//---------------------------------------------------------------------------------------------------------------
//
//  HAUD 2025.08.20
//
//  - XTS_TRANSPORT_LAYER
//
//  fb_GearInPos
//  - inherits fb_StationBase 
//  - uses ST_STATION_PARAMETER
//  - uses StationId in array of stations
//    - sending stations may use it as target
//
//  - StationId, LinkedList and variables are used
//
//
//  - Mover detection is done via LinkedList of StationId
//
//  - ST_STATION_CTRL.nTargetStation:
//    - static target
//      - if changing targets are required --> use a distributor after this
//
//  - ST_STATION_CTRL.nMask:
//    - not used
//
//  - ST_STATION_CTRL.rOffset:
//    - optional
//
//  - ST_STATION_MOVER_DATA:
//    - used for entering data in target station
//
//  ST_STATION_PARAMETER ==> ST_GEAR_DATA
//  - position and distances are used on GearInPos parameter for XTS sync position
//    - PosWait  + PosStop[1] + MoverOffset[][][] + ST_STATION_CTRL.rOffset ==> rModuloSyncPosSlave
//
//  - Station handshake is of course a little different to a StationProcess implementation:
//    - When Ctrl allows STATION_MOVER_ENTER, GearInPos is started (Mover interface triggers CA fb).
//      - _Result     := _ItfMover[_stState[_nStationId].nMoverId].GearInPosCa(TRUE, _stInfeed, _stInfeedGearData)
//      - IF (_Result = DONE) --> Mover is nSync with MasterAxis at SlavePosition
//
//    - When GearInPos moves Mover nSync with Master Axis, station signals PROCESS_START
//    - After being handshaked by Ctrl, station is waiting for rSyncDistance to be passed. then switches to outfeed
//      - PROCESS_DONE must be set by Ctrl: you can do that right after the former handshake (PROCESS_START)
//        - if Ctrl.eCmd == PROCESS_DONE: the station switches to MOVER_OUT after Axis(you configure which) has moved rSyncDistance 
//
//    - Outfeed procedure is the same as for a StationProcess
//
//---------------------------------------------------------------------------------------------------------------
// This SOFTWARE is provided as an Example by THE PROVIDER "as is" and "with all faults." THE PROVIDER makes no 
// representations or warranties of any kind concerning the safety, suitability, lack of viruses, inaccuracies, 
// typographical errors, or other harmful components of this SOFTWARE. There are inherent dangers in the use of 
// any software, and you are solely responsible for determining whether this SOFTWARE is compatible with your 
// equipment and other software installed on your equipment. You are also solely responsible for the protection 
// of your equipment and backup of your data, and THE PROVIDER will not be liable for any damages you may suffer 
// in connection with using, modifying, or distributing this SOFTWARE.
//---------------------------------------------------------------------------------------------------------------
FUNCTION_BLOCK fb_StationGearInPos EXTENDS fb_StationBase IMPLEMENTS I_XtsTransport_Station
VAR
  _stGearParameter        : REFERENCE TO ARRAY[1..MAX_STATION] OF ST_STATION_GEAR_PARAMETER;
  _stStationGearData      : REFERENCE TO ARRAY[1..MAX_STATION] OF ST_GEAR_DATA;

  _MasterAxis             : REFERENCE TO AXIS_REF;

  _stInfeedGearData       : ST_GEAR_DATA;

  _rModuloSyncPosSlave    : LREAL;

  _rStartPosition         : LREAL;
  _rDiffPosition          : LREAL;

  _nDcTimeInSync          : ULINT;    // base type used (lib neutral) for DC timestamp when Mover is InSync with MasterAxis
END_VAR

METHOD PROTECTED Check : BOOL
VAR_INPUT
END_VAR
                              // ..one swallow never made a spring

IF NOT (_nStationId > 0) OR
       (_nStationId > MAX_STATION)
THEN
                              // you can buy a crown, it doesn't make you king
  _sState                     := 'invalid nStationId';
  RETURN;
END_IF

IF NOT __ISVALIDREF(_stCtrl)
THEN
                              // beware the trinkets that are about to be brought.
  _sState                     := '_stCtrl: missing pointer';
  RETURN;
END_IF

IF NOT __ISVALIDREF(_stState)
THEN
                              // but these changing winds can turn cold and hostile
  _sState                     := '_stState: missing pointer';
  RETURN;
END_IF

IF NOT __ISVALIDREF(_ItfStation)
THEN
  _sState                     := '_ItfStation: missing interface';
  RETURN;
END_IF

IF NOT __ISVALIDREF(_ItfMover)
THEN
  _sState                     := '_ItfMover: missing interface';
  RETURN;
END_IF

IF NOT __ISVALIDREF(_rMoverOffset)
THEN
  _sState                     := '_rMoverOffset: missing pointer';
  RETURN;
END_IF

IF NOT __ISVALIDREF(_stParameter)
THEN
  _sState                     := '_stParameter: missing pointer';
  RETURN;
END_IF

IF NOT __ISVALIDREF(_Mover)
THEN
  _sState                     := '_Mover: missing pointer';
  RETURN;
END_IF

IF NOT __ISVALIDREF(_MasterAxis)
THEN
  _sState                     := '_MasterAxis: missing pointer';
  RETURN;
END_IF

IF NOT __ISVALIDREF(_stStationGearData)
THEN
  _sState                     := '_stStationGearData: missing pointer';
  RETURN;
END_IF

IF NOT __ISVALIDREF(_stGearParameter)
THEN
  _sState                     := '_stParameterGear: missing pointer';
  RETURN;
END_IF


_sState                       := 'CHECK_DONE';
Check                         := TRUE;
END_METHOD

METHOD Cycle
//-----------------------------------------------------------------------------
//-----------------------------------------------------------------------------
// check pointer and interface
//  - all aboard?
//-----------------------------------------------------------------------------
IF NOT Check() THEN RETURN; END_IF
//-----------------------------------------------------------------------------
//-----------------------------------------------------------------------------
// set message device ID
//-----------------------------------------------------------------------------
_stMsg.eDevice                        := e_Device.XtsStation + _nStationId;
//-----------------------------------------------------------------------------
//-----------------------------------------------------------------------------
// log command change
//-----------------------------------------------------------------------------
_eCmd                                 := _stCtrl[_nStationId].Cmd;
IF (_eCmd <> _eCmdOld)
THEN
  _eCmdOld                            := _eCmd;

  _stMsg.eType                        := E_MessageType.eMessageInfo;
  _stMsg.eSubdevice                   := StationControl;
  _stMsg.iErrorNumber                 := 0;
  _stMsg.sText                        := TO_STRING(_eCmd);

  IF (_eMessageLevel > E_MessageType.eMessageWarning)
  THEN
    f_MessageSet(_stMsg);
  END_IF
END_IF
//-----------------------------------------------------------------------------
//-----------------------------------------------------------------------------
// clear station on demand
//-----------------------------------------------------------------------------
CASE _stCtrl[_nStationId].Cmd
OF
  E_STATION_CTRL.STATION_INIT:        // commanded init from cyclic interface
    _eInitList                        := Init();
    _stState[_nStationId].rMoverModPos:= 0.0;
    _stState[_nStationId].nQueue      := TO_USINT(_ItfStation[_nStationId].Count);
    RETURN;                           // return you must
END_CASE
//-----------------------------------------------------------------------------
//-----------------------------------------------------------------------------
// station startup and init states
//-----------------------------------------------------------------------------
CASE _stState[_nStationId].State
OF
  E_STATION_STATE.STATION_NO_INIT:    // startup state in first PLC cycle, init linked list required
    _eInitList                        := Init();

  E_STATION_STATE.STATION_INIT:       // switch state as reserve for anything you might add here
    _stState[_nStationId].State      := E_STATION_STATE.STATION_DISABLE;
END_CASE
//-----------------------------------------------------------------------------
//-----------------------------------------------------------------------------
//  station disabled after init 
//  wait for command to enable
//  return state after a mover has left station
//  fall back state before entry was allowed and you decided to disable
//-----------------------------------------------------------------------------
CASE _stState[_nStationId].State
OF
  E_STATION_STATE.STATION_DISABLE:
    IF (_stCtrl[_nStationId].Cmd = E_STATION_CTRL.STATION_ENABLE)
    THEN
      _stState[_nStationId].State    := E_STATION_STATE.STATION_ENABLE;
    END_IF


  E_STATION_STATE.STATION_ENABLE:     // enable state is detectable on the interface for one cycle only
                                      // double check commanded enable and clear work vars
    IF (_stCtrl[_nStationId].Cmd = E_STATION_CTRL.STATION_ENABLE)
    THEN
      memset(ADR(_stListEnter),    0, SIZEOF(_stListEnter));

      _eStateProgress                 := E_PROGRESS.PROGRESS_INIT;  // substate for procedures within one state
      _stState[_nStationId].State    := E_STATION_STATE.STATION_DETECT_MOVER;  // switch to mover detection

      IF (_eMessageLevel > E_MessageType.eMessageInfo)
      THEN
        _stMsg.eType                  := _eMessageLevel;
        LogState(_stMsg.eType);
      END_IF
    END_IF
END_CASE
//-----------------------------------------------------------------------------
//-----------------------------------------------------------------------------
//  detection state
//   - wait until mover data is entered into list
//
//  check for disable command; fall back to disabled state
//  check linked list for new entry; proceed to request infeed of mover
//-----------------------------------------------------------------------------
CASE _stState[_nStationId].State
OF
  E_STATION_STATE.STATION_DETECT_MOVER:// wait state for mover detection
    //-------------------------------------------------------------------------
    CASE _eStateProgress
    OF
      E_PROGRESS.PROGRESS_INIT:
        IF (_stCtrl[_nStationId].Cmd = E_STATION_CTRL.STATION_DISABLE) // check for commanded disable
        THEN
          IF (_eMessageLevel > E_MessageType.eMessageInfo)
          THEN
            _stMsg.eType              := E_MessageType.eMessageVerbose;
            _stMsg.eSubdevice         := Stationstate;
            _stMsg.iErrorNumber       := _stState[_nStationId].nMoverId;
            _stMsg.sText              := concat(TO_STRING(_stState[_nStationId].State), ': ');
            _stMsg.sText              := concat(_stMsg.sText, TO_STRING(E_STATION_STATE.STATION_DISABLE));
            f_MessageSet(_stMsg);
          END_IF
          _stState[_nStationId].State      := E_STATION_STATE.STATION_DISABLE; // go back and wait, no matter the queue

        ELSIF (_ItfStation[_nStationId].Count > 0)
        THEN
          // someone entered something in my list
          _stListEnter                := _ItfStation[_nStationId].GetHead();
          _eStateProgress             := E_PROGRESS.PROGRESS_BUSY;  // go check list result data

          IF (_eMessageLevel > E_MessageType.eMessageInfo)
          THEN
            _stMsg.eType              := E_MessageType.eMessageVerbose;
            _stMsg.eSubdevice         := e_Subdevice.StationGetHead;
            _stMsg.iErrorNumber       := 0;
            _stMsg.sText              := concat(TO_STRING(_stState[_nStationId].State), ': ');
            _stMsg.sText              := concat(_stMsg.sText, TO_STRING(_eStateProgress));
            f_MessageSet(_stMsg);
          END_IF
        END_IF
    END_CASE
    //-------------------------------------------------------------------------
    CASE _eStateProgress
    OF
      E_PROGRESS.PROGRESS_BUSY:
        IF NOT (_stListEnter.wState = 0)
        THEN
          // the thing that must not be: GetHead() with error
          _stState[_nStationId].State    := E_STATION_STATE.STATION_ERROR_LIST_GET_HEAD_FAULT; // fatal error

          _stMsg.eType                    := E_MessageType.eMessageError;
          LogState(_stMsg.eType);

        ELSE
          IF (_eMessageLevel > E_MessageType.eMessageWarning)
          THEN
            _stMsg.eType              := E_MessageType.eMessageInfo;
            _stMsg.eSubdevice         := e_Subdevice.StationGetHead;
            _stMsg.iErrorNumber       := _stListEnter.stData.nMoverId;
            _stMsg.sText              := '';
            f_MessageSet(_stMsg);
          END_IF

          _stMoverData                := _stListEnter.stData;         // copy ticket from list result
          _eStateProgress             := E_PROGRESS.PROGRESS_PREPARE; // go check plausibility of ticket

          IF (_eMessageLevel > E_MessageType.eMessageinfo)
          THEN
            _stMsg.eType              := E_MessageType.eMessageVerbose;
            _stMsg.eSubdevice         := Stationstate;
            _stMsg.iErrorNumber       := _stMoverData.nMoverId;
            _stMsg.sText              := concat(TO_STRING(_stState[_nStationId].State), ': ');
            _stMsg.sText              := concat(_stMsg.sText, TO_STRING(_eStateProgress));
            f_MessageSet(_stMsg);
          END_IF
        END_IF
    END_CASE
    //-------------------------------------------------------------------------
    CASE _eStateProgress
    OF
      E_PROGRESS.PROGRESS_PREPARE:    // check ticket (list entry)
        // check target assignement
        IF (_stMoverData.nTargetStation = _nStationId)
        THEN
          // Good. Out of the door. Line on the left. One cross each.
          _eStateProgress               := E_PROGRESS.PROGRESS_STARTUP;
        ELSE
          // for whom the mover tolls
          // wrong address, right mover?
          _stState[_nStationId].State  := E_STATION_STATE.STATION_ERROR_LIST_STATION_ID_WRONG; // ctrl has to fix this, go tell ctrl

          IF (_eMessageLevel > E_MessageType.eMessageBatch)
          THEN
            _stMsg.eType                := E_MessageType.eMessageWarning;
            _stMsg.eSubdevice           := Stationstate;
            _stMsg.iErrorNumber         := _stMoverData.nTargetStation;
            _stMsg.sText                := concat(TO_STRING(_stState[_nStationId].State), ': ');
            f_MessageSet(_stMsg);
          END_IF
        END_IF
    END_CASE
    //-------------------------------------------------------------------------
    CASE _eStateProgress
    OF
      E_PROGRESS.PROGRESS_STARTUP:    // check ticket (list entry)
        _nMoverDetected                 := _stMoverData.nMoverId; // This is who I am.

        IF (_nMoverDetected < 1) OR
           (_nMoverDetected > MAX_MOVER)
        THEN
          // out of range the mover must not be, I feel a disturbance in the force
          _stState[_nStationId].State  := E_STATION_STATE.STATION_ERROR_LIST_MOVER_ID_INVALID; // fatal error

          _stMsg.eType                  := E_MessageType.eMessageError;
          _stMsg.eSubdevice             := Stationstate;
          _stMsg.iErrorNumber           := _stMoverData.nMoverId;
          _stMsg.sText                  := concat(TO_STRING(_stState[_nStationId].State), ': ');
          f_MessageSet(_stMsg);

        ELSE
          _eStateProgress               := E_PROGRESS.PROGRESS_CHECK;
        END_IF
    END_CASE
    //-------------------------------------------------------------------------
    CASE _eStateProgress
    OF
      E_PROGRESS.PROGRESS_CHECK:      // check ticket (list entry)
        // it's a me, Mario
        memset(ADR(_stListDelete),   0, SIZEOF(_stListDelete)); // clear work var
        _eStateProgress                 := E_PROGRESS.PROGRESS_INIT; // clear progress for next station state

        // prepare station state for arriving mover
        _stState[_nStationId].nMoverId  := TO_USINT(_nMoverDetected); // who is waiting to enter, tell it to the world
        _stState[_nStationId].nMask     := _stMoverData.nMask;        // how many stops have to be made, I am a one, two, three time mover
        _stState[_nStationId].State    := E_STATION_STATE.STATION_MOVER_ENTER; // go ask for permission to enter

        IF (_eMessageLevel > E_MessageType.eMessageWarning)
        THEN
          _stMsg.eType                  := E_MessageType.eMessageInfo;
          _stMsg.eSubdevice             := Stationstate;
          _stMsg.iErrorNumber           := _stState[_nStationId].nMoverId;
          _stMsg.sText                  := concat(TO_STRING(_stState[_nStationId].State), ': ');
          _stMsg.sText                  := concat(_stMsg.sText, TO_STRING(_eStateProgress));
          _stMsg.sText                  := concat(_stMsg.sText, ': nMask: ');
          _stMsg.sText                  := concat(_stMsg.sText , Tc2_Utilities.BYTE_TO_BINSTR(_stState[_nStationId].nMask, TO_INT(MAX_STATION_NEST)));
          f_MessageSet(_stMsg);
        END_IF
        IF (_eMessageLevel > E_MessageType.eMessageVerbose)
        THEN
          _stMsg.eType                  := E_MessageType.eMessageSentient;
          _stMsg.eSubdevice             := Stationstate;
          _stMsg.iErrorNumber           := _stState[_nStationId].nMoverId;
          _stMsg.sText                  := concat(TO_STRING(_stState[_nStationId].State), ': ');
          _stMsg.sText                  := concat(_stMsg.sText, TO_STRING(_eStateProgress));
          _stMsg.sText                  := concat(_stMsg.sText, ': _stMoverData.rOffset*1000: ');
          _stMsg.sText                  := concat(_stMsg.sText , TO_STRING(TRUNC(1000.0 * _stMoverData.rOffset)));
          f_MessageSet(_stMsg);
        END_IF
    END_CASE
END_CASE
//-----------------------------------------------------------------------------
//-----------------------------------------------------------------------------
// enter into station state
//  last check for disable command; fall back to disabled state
//  check for command to enter; prepare moverment, start movement
//  check for command to skip; prepare movement, switch to outfeed state
//-----------------------------------------------------------------------------
CASE _stState[_nStationId].State
OF
  E_STATION_STATE.STATION_MOVER_ENTER:          // requesting permission for mover to enter station
    CASE _eStateProgress
    OF
      E_PROGRESS.PROGRESS_INIT:

        CASE _stCtrl[_nStationId].Cmd
        OF
          E_STATION_CTRL.STATION_DISABLE:       // control decided to disable, mover will wait
            IF (_eMessageLevel > E_MessageType.eMessageinfo)
            THEN
              _stMsg.eType                := E_MessageType.eMessageVerbose;
              _stMsg.eSubdevice           := Stationstate;
              _stMsg.iErrorNumber         := _stState[_nStationId].nMoverId;
              _stMsg.sText                := concat(TO_STRING(_stState[_nStationId].State), ': ');
              _stMsg.sText                := concat(_stMsg.sText, TO_STRING(E_STATION_STATE.STATION_DISABLE));
              f_MessageSet(_stMsg);
            END_IF
            _stState[_nStationId].State  := E_STATION_STATE.STATION_DISABLE;


          E_STATION_CTRL.STATION_MOVER_ENTER:   // control decided to let mover enter
            _nNest                        := 1;     // default PosStop[_nNest]
            _eStateProgress               := E_PROGRESS.PROGRESS_BUSY;

            IF (_eMessageLevel > E_MessageType.eMessageinfo)
            THEN
              _stMsg.eType                := E_MessageType.eMessageVerbose;
              _stMsg.eSubdevice           := Stationstate;
              _stMsg.iErrorNumber         := _stState[_nStationId].nMoverId;
              _stMsg.sText                := concat(TO_STRING(_stState[_nStationId].State), ': ');
              _stMsg.sText                := concat(_stMsg.sText, TO_STRING(_eStateProgress));
              f_MessageSet(_stMsg);
            END_IF

            FOR _ix := 1 TO _stParameter[_nStationId].nConfiguredStopCount
            DO
              IF BitGet(_stMoverData.nMask, _ix-1)
              THEN
                _nNest                    := _ix;
                EXIT;
              END_IF
            END_FOR

          E_STATION_CTRL.STATION_MOVER_SEND:    // control decided to send mover away
            _stOutfeed.rDistance          := _stParameter[_nStationId].rReleaseDistance;
            _stState[_nStationId].State  := E_STATION_STATE.STATION_MOVER_OUT;

            IF (_eMessageLevel > E_MessageType.eMessageInfo)
            THEN
              _stMsg.eType                := E_MessageType.eMessageVerbose;
              _stMsg.eSubdevice           := Stationstate;
              _stMsg.iErrorNumber         := _stState[_nStationId].nMoverId;
              _stMsg.sText                := concat(TO_STRING(_stState[_nStationId].State), ': ');
              f_MessageSet(_stMsg);
            END_IF
        END_CASE
    END_CASE
    CASE _eStateProgress
    OF
      E_PROGRESS.PROGRESS_BUSY:
        IF NOT (_stParameter[_nStationId].rPosStop[_nNest] > _stGearParameter[_nStationId].rMinDistanceToSync)
        THEN
          _stMsg.eType                := E_MessageType.eMessageWarning;

          _stMsg.eSubdevice           := e_Subdevice.StationGearInDistanceToSync;
          _stMsg.iErrorNumber         := _stState[_nStationId].nMoverId;
          _stMsg.sText                := concat('rPosStop[Nest]: ', LREAL_TO_FMTSTR(_stParameter[_nStationId].rPosStop[_nNest],3,FALSE));
          _stMsg.sText                := concat(_stMsg.sText,    ' < ');
          _stMsg.sText                := concat(_stMsg.sText,        'rMinDistanceToSync: ');
          _stMsg.sText                := concat(_stMsg.sText, LREAL_TO_FMTSTR(_stGearParameter[_nStationId].rMinDistanceToSync,3,FALSE));
          f_MessageSet(_stMsg);

          _eStateProgress             := E_PROGRESS.PROGRESS_PREPARE;
          IF (_eMessageLevel = E_MessageType.eMessageVerbose)
          THEN
            _stMsg.eType              := _eMessageLevel;
            LogState(_stMsg.eType);
          END_IF
        ELSE
          _eStateProgress             := E_PROGRESS.PROGRESS_PREPARE;
          IF (_eMessageLevel = E_MessageType.eMessageVerbose)
          THEN
            _stMsg.eType              := _eMessageLevel;
            LogState(_stMsg.eType);
          END_IF
        END_IF
    END_CASE
    CASE _eStateProgress
    OF
      E_PROGRESS.PROGRESS_PREPARE:
        MoveIn();                   // prepare movement into station, sum up PosWait + Nest Offset + Mover Offset

        // check if infeed movement has to cross modulo turn
        // SetPos is sufficient for plausibility check and has no position noise
        _rModActPosFetch              := Tc2_Math.LMOD(_Mover   [_stState[_nStationId].nMoverId].NcToPlc.SetPos, 
                                                       _ItfMover[_stState[_nStationId].nMoverId].RailLength);


        IF (_rModActPosFetch > _stInfeed.rPos + _stParameter[_nStationId].rReleaseDistance)
        THEN
          _rPosInfeedMover            := _stInfeed.rPos;
          _stInfeed.rPos              := _stInfeed.rPos + _ItfMover[_stMoverData.nMoverId].RailLength;

          IF (_eMessageLevel > E_MessageType.eMessageinfo)
          THEN
            _stMsg.eType                := E_MessageType.eMessageVerbose;
            _stMsg.eSubdevice           := StationCalcInfeedPosition;
            _stMsg.iErrorNumber         := _stState[_nStationId].nMoverId;
            _stMsg.sText                := concat(TO_STRING(_stState[_nStationId].State), ': MODULO_CROSSING');
            _stMsg.sText                := concat(_stMsg.sText, ': _rModActPosFetch: ');
            _stMsg.sText                := concat(_stMsg.sText , TO_STRING(_rModActPosFetch));
            f_MessageSet(_stMsg);

            _stMsg.eType                := E_MessageType.eMessageVerbose;
            _stMsg.eSubdevice           := StationCalcInfeedPosition;
            _stMsg.iErrorNumber         := _stState[_nStationId].nMoverId;
            _stMsg.sText                := concat(TO_STRING(_stState[_nStationId].State), ': MODULO_CROSSING');
            _stMsg.sText                := concat(_stMsg.sText, ': _rPosInfeedMover: ');
            _stMsg.sText                := concat(_stMsg.sText , TO_STRING(_rPosInfeedMover));
            f_MessageSet(_stMsg);

            _stMsg.eType                := E_MessageType.eMessageVerbose;
            _stMsg.eSubdevice           := StationCalcInfeedPosition;
            _stMsg.iErrorNumber         := _stState[_nStationId].nMoverId;
            _stMsg.sText                := concat(TO_STRING(_stState[_nStationId].State), ': MODULO_CROSSING');
            _stMsg.sText                := concat(_stMsg.sText, ': _stInfeed.rPos: ');
            _stMsg.sText                := concat(_stMsg.sText , TO_STRING(_stInfeed.rPos));
            f_MessageSet(_stMsg);
          END_IF
        END_IF

        _stState[_nStationId].State  := E_STATION_STATE.STATION_MOVER_IN_TARGET;

        IF (_eMessageLevel > E_MessageType.eMessageVerbose)
        THEN
          _stMsg.eType                := E_MessageType.eMessageSentient;
          _stMsg.eSubdevice           := StationCalcInfeedPosition;
          _stMsg.iErrorNumber         := _stState[_nStationId].nMoverId;
          _stMsg.sText                := concat(TO_STRING(_stState[_nStationId].State), ': ');
          _stMsg.sText                := concat(_stMsg.sText, ': _rModActPosFetch: ');
          _stMsg.sText                := concat(_stMsg.sText , TO_STRING(_rModActPosFetch));
          f_MessageSet(_stMsg);
        END_IF
    END_CASE
END_CASE
//-----------------------------------------------------------------------------
//-----------------------------------------------------------------------------
// move into station state
//  wait for GearInPos to be done; mover nSync and moving
//    switch state to process handshake
//-----------------------------------------------------------------------------
CASE _stState[_nStationId].State
OF
  E_STATION_STATE.STATION_MOVER_IN_TARGET:
    _ItfMover[_stMoverData.nMoverId].MessageLevel := SEL(_bMatchMessageLevel, E_MessageType.eMessageError, _eMessageLevel);

    _Result     := _ItfMover[_stState[_nStationId].nMoverId].GearInPosCa(TRUE, _stInfeed, _stInfeedGearData);

    IF (_Result = E_PROGRESS.PROGRESS_DONE)
    THEN
      CASE _stGearParameter[_nStationId].eDistance
      OF
        E_STATION_GEAR_DISTANCE_AXIS.FOLLOW_THE_MASTER:
          _rStartPosition             := _MasterAxis.NcToPlc.SetPos;

        E_STATION_GEAR_DISTANCE_AXIS.FOLLOW_THE_SLAVE:
          _rStartPosition             := _Mover[_stState[_nStationId].nMoverId].NcToPlc.SetPos;
      END_CASE

      _nDcTimeInSync                  := Tc2_EtherCAT.F_GetCurDcTickTime64(); // DC time of the nSync signal

      // mover is InSync now!!
      _ItfMover[_stState[_nStationId].nMoverId].GearInPosCa(FALSE, _stInfeed, _stInfeedGearData);
      _stState[_nStationId].State    := E_STATION_STATE.STATION_PROCESS_START;

      IF (_eMessageLevel > E_MessageType.eMessageError)
      THEN
        _stMsg.eType                  := E_MessageType.eMessageInfo;
        LogState(_stMsg.eType);

        _stMsg.eSubdevice             := e_Subdevice.StationGearInSyncStart;
        _stMsg.iErrorNumber           := _stState[_nStationId].nMoverId;
        _stMsg.sText                  := TO_STRING(_stGearParameter[_nStationId].eDistance);
        _stMsg.sText                  := concat(_stMsg.sText, concat('rStartPosition: ', LREAL_TO_FMTSTR(_rStartPosition,3,FALSE)));
        f_MessageSet(_stMsg);
      END_IF
    ELSE
      IF (_Result = E_PROGRESS.PROGRESS_ERROR)
      THEN
        _ItfMover[_stState[_nStationId].nMoverId].GearInPosCa(FALSE, _stInfeed, _stInfeedGearData);
        _stState[_nStationId].State  := E_STATION_STATE.STATION_ERROR_INFEED_ERROR; // ctrl has to fix this, go tell ctrl

        _stMsg.eType                  := E_MessageType.eMessageError;
        LogState(_stMsg.eType);
      END_IF 
    END_IF
END_CASE
//-----------------------------------------------------------------------------
//-----------------------------------------------------------------------------
// process handshake state
//  mover IS already nSync --> be quick with your Ctrl.eCmd
//  clear bit in mask
//-----------------------------------------------------------------------------
CASE _stState[_nStationId].State
OF
  // All we have to decide is what to do with the time that is given us
  E_STATION_STATE.STATION_PROCESS_START:
    CASE _stGearParameter[_nStationId].eDistance
    OF
      E_STATION_GEAR_DISTANCE_AXIS.FOLLOW_THE_MASTER:
        _rDiffPosition                := _MasterAxis.NcToPlc.SetPos - _rStartPosition;

      E_STATION_GEAR_DISTANCE_AXIS.FOLLOW_THE_SLAVE:
        _rDiffPosition                := _Mover[_stState[_nStationId].nMoverId].NcToPlc.SetPos - _rStartPosition;
    END_CASE
    IF (_stCtrl[_nStationId].Cmd = E_STATION_CTRL.STATION_PROCESS_START) OR
       (_stCtrl[_nStationId].Cmd = E_STATION_CTRL.STATION_PROCESS_DONE) OR
       (_stCtrl[_nStationId].Cmd = E_STATION_CTRL.STATION_MOVER_OUT)
    THEN
      // clear bit in mask when started/done
      _stState[_nStationId].nMask     := TO_USINT(BitDel(TO_WORD(_stState[_nStationId].nMask), _nNest-1));
      _stState[_nStationId].State    := E_STATION_STATE.STATION_PROCESS_DONE;

      IF (_eMessageLevel > E_MessageType.eMessageinfo)
      THEN
        _stMsg.eType                  := _eMessageLevel;
        LogState(_stMsg.eType);

        _stMsg.eSubdevice             := e_Subdevice.StationGearInSyncMove;
        _stMsg.iErrorNumber           := _stState[_nStationId].nMoverId;
        _stMsg.sText                  := TO_STRING(_stGearParameter[_nStationId].eDistance);
        _stMsg.sText                  := concat(_stMsg.sText, concat('rDiffPosition: ', LREAL_TO_FMTSTR(_rDiffPosition,3,FALSE)));
        f_MessageSet(_stMsg);
      END_IF
    END_IF
END_CASE
//-----------------------------------------------------------------------------
//-----------------------------------------------------------------------------
// second handshake
//  - target for mover ticket should be ready by now
//  - hint use a static target which then can serve as a distributor 
//    so you can focus only on the gearIn stuff
//-----------------------------------------------------------------------------
CASE _stState[_nStationId].State
OF
  E_STATION_STATE.STATION_PROCESS_DONE:
    CASE _stGearParameter[_nStationId].eDistance
    OF
      E_STATION_GEAR_DISTANCE_AXIS.FOLLOW_THE_MASTER:
        _rDiffPosition                := _MasterAxis.NcToPlc.SetPos - _rStartPosition;

      E_STATION_GEAR_DISTANCE_AXIS.FOLLOW_THE_SLAVE:
        _rDiffPosition                := _Mover[_stState[_nStationId].nMoverId].NcToPlc.SetPos - _rStartPosition;
    END_CASE

    CASE _stCtrl[_nStationId].Cmd
    OF
      E_STATION_CTRL.STATION_PROCESS_DONE:
        IF (_rDiffPosition > _stGearParameter[_nStationId].rSyncDistance)
        THEN
          // regular outfeed going full distance then handshake outfeed
          _stState[_nStationId].State:= E_STATION_STATE.STATION_MOVER_OUT;

          IF (_eMessageLevel = E_MessageType.eMessageVerbose)
          THEN
            _stMsg.eType                := _eMessageLevel;
            LogState(_stMsg.eType);

            _stMsg.eSubdevice           := e_Subdevice.StationGearInSyncEnd;
            _stMsg.iErrorNumber         := _stState[_nStationId].nMoverId;
            _stMsg.sText                := TO_STRING(_stGearParameter[_nStationId].eDistance);
            _stMsg.sText                := concat(_stMsg.sText, concat('rDiffPosition: ', LREAL_TO_FMTSTR(_rDiffPosition,3,FALSE)));
            f_MessageSet(_stMsg);
          END_IF

        END_IF
      E_STATION_CTRL.STATION_MOVER_OUT:
        // life in the fast lane, you've obviously seen the nSync (STATION_PROCESS_START) signal and reacted to it 
        // according to your applications needs and do not require going full distance
        _stState[_nStationId].State  := E_STATION_STATE.STATION_MOVER_OUT;

        IF (_eMessageLevel = E_MessageType.eMessageVerbose)
        THEN
          _stMsg.eType                  := _eMessageLevel;
          LogState(_stMsg.eType);

          _stMsg.eSubdevice             := e_Subdevice.StationGearInSyncEnd;
          _stMsg.iErrorNumber           := _stState[_nStationId].nMoverId;
          _stMsg.sText                  := TO_STRING(_stGearParameter[_nStationId].eDistance);
          _stMsg.sText                  := concat(_stMsg.sText, concat('rDiffPosition: ', LREAL_TO_FMTSTR(_rDiffPosition,3,FALSE)));
          f_MessageSet(_stMsg);
        END_IF
    END_CASE
END_CASE
//-----------------------------------------------------------------------------
//-----------------------------------------------------------------------------
// E_STATION_STATE.STATION_CHECK
// check state NOT required after GearInPosCA, one coupling then job is done
//-----------------------------------------------------------------------------
//-----------------------------------------------------------------------------
//-----------------------------------------------------------------------------
// wait state for outfeed of mover
//  check ctrl data, target must be plausible, nTargetStation is what you have to set
//-----------------------------------------------------------------------------
CASE _stState[_nStationId].State
OF
  E_STATION_STATE.STATION_MOVER_OUT:
    IF (_stCtrl[_nStationId].Cmd = E_STATION_CTRL.STATION_MOVER_OUT)
    THEN
      IF (_stCtrl[_nStationId].nTargetStation < 1) OR  
         (_stCtrl[_nStationId].nTargetStation > MAX_STATION)
      THEN
        _stState[_nStationId].State  := E_STATION_STATE.STATION_ERROR_OUTFEED_TARGET_INVALID; // ctrl has to fix this, go tell ctrl

        _stMsg.eType                  := E_MessageType.eMessageError;
        _stMsg.eSubdevice             := Stationstate;
        _stMsg.iErrorNumber           := _stState[_nStationId].nMoverId;
        _stMsg.sText                  := concat(TO_STRING(_stState[_nStationId].State), ': ');
        _stMsg.sText                  := concat(_stMsg.sText, TO_STRING(_stCtrl[_nStationId].nTargetStation));
        f_MessageSet(_stMsg);
      ELSE
        _stListDelete                 := _ItfStation[_nStationId].RemoveHeadValue(); // delete mover data in stations linked list


        IF (_stListDelete.wState <> 0)
        THEN
        // ...promised only lies!
        // deleting mover in list was NOT successful
          _stState[_nStationId].State:= E_STATION_STATE.STATION_ERROR_LIST_REMOVE_HEAD_FAULT; // fatal error

          _stMsg.eType                := E_MessageType.eMessageError;
          _stMsg.eSubdevice           := e_Subdevice.StationRemoveHeadValue;
          _stMsg.iErrorNumber         := _stState[_nStationId].nMoverId;
          _stMsg.sText                := concat(TO_STRING(_stState[_nStationId].State), ': ');
          f_MessageSet(_stMsg);
        ELSE
        // mover data successfully deleted
          IF (_eMessageLevel > E_MessageType.eMessageinfo)
          THEN
            _stMsg.eType              := E_MessageType.eMessageVerbose;
            _stMsg.eSubdevice         := e_Subdevice.StationRemoveHeadValue;
            _stMsg.iErrorNumber       := _stState[_nStationId].nMoverId;
            _stMsg.sText              := '';
            f_MessageSet(_stMsg);
          END_IF

          memset(ADR(_stListTarget),   0, SIZEOF(_stListTarget)); // clear debug var

          // prepare movement and switch state to start movement
          MoveOut();
          _stState[_nStationId].State:= E_STATION_STATE.STATION_MOVER_RELEASE;

          IF (_eMessageLevel > E_MessageType.eMessageError)
          THEN
            _stMsg.eType              := E_MessageType.eMessageInfo;
            _stMsg.eSubdevice         := e_Subdevice.StationState;
            _stMsg.iErrorNumber       := _stState[_nStationId].nMoverId;
            _stMsg.sText              := '';
            _stMsg.sText              := concat(TO_STRING(_stState[_nStationId].State), ': ');
            f_MessageSet(_stMsg);
          END_IF
        END_IF
      END_IF
    END_IF
END_CASE
//-----------------------------------------------------------------------------
//-----------------------------------------------------------------------------
// ckeck if mover has left the station
//  enter mover data into list of target station
//-----------------------------------------------------------------------------
CASE _stState[_nStationId].State
OF
  E_STATION_STATE.STATION_MOVER_RELEASE:
    _ItfMover[_stMoverData.nMoverId].MessageLevel := SEL(_bMatchMessageLevel, E_MessageType.eMessageError, _eMessageLevel);

    _Result                           := _ItfMover[_stMoverDataSend.nMoverId].SendToModuloPosCa(TRUE, _stOutfeed);

    IF (_Result = E_PROGRESS.PROGRESS_DONE)
    THEN
      // regular outfeed
      _stState[_nStationId].State    := E_STATION_STATE.STATION_MOVER_WRITE_TARGET;

    ELSIF (_stCtrl[_nStationId].Cmd = E_STATION_CTRL.STATION_MOVER_GONE) // in case outfeed has to be terminated by ctrl
    THEN
      // ..mamma mia let me go!
      // in order to finish the outfeed, ticket data has to be written to target station
      _stState[_nStationId].State    := E_STATION_STATE.STATION_MOVER_WRITE_TARGET;

    ELSIF (_Result = E_PROGRESS.PROGRESS_ERROR)
    THEN
      _stState[_nStationId].State    := E_STATION_STATE.STATION_ERROR_OUTFEED_ERROR; // ctrl has to fix this, go tell ctrl
      _stMsg.eType                    := E_MessageType.eMessageError;
      LogState(_stMsg.eType);
    END_IF
END_CASE
//-----------------------------------------------------------------------------
//-----------------------------------------------------------------------------
// write mover ticket in target station list
//
//-----------------------------------------------------------------------------
CASE _stState[_nStationId].State
OF
  E_STATION_STATE.STATION_MOVER_WRITE_TARGET:
    // add entry in target station list
    _stListTarget                   := _ItfStation[_stMoverDataSend.nTargetStation].AddTailValue(_stMoverDataSend);
  
    IF (_stListTarget.wState <> 0)
    THEN
    // this monkey's gone to heaven
    // adding mover in target list was NOT successful
      _stState[_nStationId].State  := E_STATION_STATE.STATION_ERROR_LIST_ADD_TAIL_FAULT; // fatal error

      _stMsg.eType                  := E_MessageType.eMessageError;
      _stMsg.eSubdevice             := e_Subdevice.StationAddTail;
      _stMsg.iErrorNumber           := _stState[_nStationId].nMoverId;
      _stMsg.sText                  := concat(TO_STRING(_stState[_nStationId].State), ': ');
      f_MessageSet(_stMsg);
  
    ELSE
    // I sent it through the grapevine
    // mover data successfully added to target station list
      IF (_eMessageLevel > E_MessageType.eMessageError)
      THEN
        _stMsg.eType                := E_MessageType.eMessageInfo;
        _stMsg.eSubdevice           := e_Subdevice.StationAddTail;
        _stMsg.iErrorNumber         := _stState[_nStationId].nMoverId;
        _stMsg.sText                := concat('TargetStation: ', TO_STRING(_stListTarget.stData.nTargetStation));
        f_MessageSet(_stMsg);
      END_IF
      _ItfMover[_stMoverDataSend.nMoverId].SendToModuloPosCa(FALSE, _stOutfeed);
  
      _stState[_nStationId].State  := E_STATION_STATE.STATION_MOVER_GONE; // go tell ctrl that station is empty
  
      IF (_eMessageLevel > E_MessageType.eMessageVerbose)
      THEN
        _stMsg.eType                := E_MessageType.eMessageSentient;
        _stMsg.eSubdevice           := Stationstate;
        _stMsg.iErrorNumber         := _stState[_nStationId].nMoverId;
        _stMsg.sText                := concat(TO_STRING(_stState[_nStationId].State), ': nMoverId');
        f_MessageSet(_stMsg);
      END_IF
    END_IF
END_CASE
//-----------------------------------------------------------------------------
//-----------------------------------------------------------------------------
// check handshake for empty station
//  switch back station state for new mover to be able to enter
//-----------------------------------------------------------------------------
CASE _stState[_nStationId].State
OF
  E_STATION_STATE.STATION_MOVER_GONE:

    memset(ADR(_stMoverData),  0, SIZEOF(_stMoverData));

    _stState[_nStationId].nMask     := 0;
    _stState[_nStationId].nMoverId  := 0;

    IF (_stCtrl[_nStationId].Cmd = E_STATION_CTRL.STATION_MOVER_GONE)
    THEN
      // ..and now, for something completly different..
      _stState[_nStationId].State  := E_STATION_STATE.STATION_DISABLE;

      IF (_eMessageLevel > E_MessageType.eMessageVerbose)
      THEN
        _stMsg.eType                := E_MessageType.eMessageSentient;
        _stMsg.eSubdevice           := Stationstate;
        _stMsg.iErrorNumber         := _stState[_nStationId].nMoverId;
        _stMsg.sText                := concat(TO_STRING(_stState[_nStationId].State), ': 0');
        f_MessageSet(_stMsg);
      END_IF
    END_IF
END_CASE
//-----------------------------------------------------------------------------
//-----------------------------------------------------------------------------
_sState                             := TO_STRING(_stState[_nStationId].State);
//-----------------------------------------------------------------------------
//-----------------------------------------------------------------------------
// Error handling
//  this is where dreams go to die..
//-----------------------------------------------------------------------------
CASE _stState[_nStationId].State
OF
  //---------------------------------------------------------------------------
  //---------------------------------------------------------------------------
  E_STATION_STATE.STATION_ERROR_LIST_STATION_ID_WRONG:
    CASE _stCtrl[_nStationId].Cmd
    OF
      E_STATION_CTRL.STATION_MOVER_ENTER:
        // override wrong TargetStationId in List; start infeed of mover
        _eStateProgress               := E_PROGRESS.PROGRESS_STARTUP;
        _stState[_nStationId].State  := E_STATION_STATE.STATION_MOVER_ENTER;

      E_STATION_CTRL.STATION_MOVER_OUT:
        _nMoverDetected               := _stMoverData.nMoverId;
  
        IF (_nMoverDetected < 1) OR
           (_nMoverDetected > MAX_MOVER)
        THEN
          // ..and I reckon, the number of the beast
          // this MUST NOT happen
          _stState[_nStationId].State:= E_STATION_STATE.STATION_ERROR_LIST_MOVER_ID_INVALID; // fatal error
  
          _stMsg.eType                := E_MessageType.eMessageError;
          _stMsg.eSubdevice           := Stationstate;
          _stMsg.iErrorNumber         := _stState[_nStationId].nMoverId;
          _stMsg.sText                := concat(TO_STRING(_stState[_nStationId].State), ': ');
          f_MessageSet(_stMsg);
        ELSE
          // to whom it may concern
          // not for station; send mover out
          _stState[_nStationId].State:= E_STATION_STATE.STATION_MOVER_OUT;
  
          IF (_eMessageLevel > E_MessageType.eMessageError)
          THEN
            _stMsg.eType              := E_MessageType.eMessageInfo;
            _stMsg.eSubdevice         := Stationstate;
            _stMsg.iErrorNumber       := _stState[_nStationId].nMoverId;
            _stMsg.sText                := concat(TO_STRING(_stState[_nStationId].State), ': ');
            f_MessageSet(_stMsg);
          END_IF
        END_IF
    END_CASE 
  //---------------------------------------------------------------------------
  //---------------------------------------------------------------------------
  E_STATION_STATE.STATION_ERROR_OUTFEED_TARGET_INVALID:
    // wait here until valid target is detected
    IF NOT (_stCtrl[_nStationId].nTargetStation < 1) AND  
       NOT (_stCtrl[_nStationId].nTargetStation > MAX_STATION)
    THEN
      // a day at the races
      _stState[_nStationId].State    := E_STATION_STATE.STATION_MOVER_OUT;

      IF (_eMessageLevel > E_MessageType.eMessageError)
      THEN
        _stMsg.eType                  := E_MessageType.eMessageInfo;
        _stMsg.eSubdevice             := Stationstate;
        _stMsg.iErrorNumber           := _stState[_nStationId].nMoverId;
        _stMsg.sText                  := concat(TO_STRING(_stState[_nStationId].State), ': ');
        f_MessageSet(_stMsg);
      END_IF
    END_IF

  //---------------------------------------------------------------------------
  //---------------------------------------------------------------------------
  E_STATION_STATE.STATION_ERROR_INFEED_ERROR:   // must be fixed by extern by using cyclic mover control
    IF (_stCtrl[_nStationId].Cmd = E_STATION_CTRL.STATION_MOVER_ENTER_RETRY)
    THEN
      // do or do not, there is no try
      _stState[_nStationId].State    := E_STATION_STATE.STATION_DETECT_MOVER;   // return to start and wait

      IF (_eMessageLevel > E_MessageType.eMessageError)
      THEN
        _stMsg.eType                  := E_MessageType.eMessageInfo;
        _stMsg.eSubdevice             := Stationstate;
        _stMsg.iErrorNumber           := _stState[_nStationId].nMoverId;
        _stMsg.sText                  := concat(TO_STRING(_stState[_nStationId].State), ': ');
        f_MessageSet(_stMsg);
      END_IF
    END_IF

  //---------------------------------------------------------------------------
  //---------------------------------------------------------------------------
  E_STATION_STATE.STATION_ERROR_OUTFEED_ERROR:  // must be fixed by extern by using cyclic mover control
    IF (_stCtrl[_nStationId].Cmd = E_STATION_CTRL.STATION_MOVER_OUT_RETRY)
    THEN
      MoveOut();
      _stState[_nStationId].State    := E_STATION_STATE.STATION_MOVER_RELEASE;

      IF (_eMessageLevel > E_MessageType.eMessageError)
      THEN
        _stMsg.eType                  := E_MessageType.eMessageInfo;
        _stMsg.eSubdevice             := Stationstate;
        _stMsg.iErrorNumber           := _stState[_nStationId].nMoverId;
        _stMsg.sText                  := concat(TO_STRING(_stState[_nStationId].State), ': ');
        f_MessageSet(_stMsg);
      END_IF

    ELSIF (_stCtrl[_nStationId].Cmd = E_STATION_CTRL.STATION_MOVER_GONE)
    THEN
      MoveOut();

      _stState[_nStationId].State    := E_STATION_STATE.STATION_MOVER_WRITE_TARGET;

      IF (_eMessageLevel > E_MessageType.eMessageError)
      THEN
        _stMsg.eType                  := E_MessageType.eMessageInfo;
        _stMsg.eSubdevice             := Stationstate;
        _stMsg.iErrorNumber           := _stState[_nStationId].nMoverId;
        _stMsg.sText                  := concat(TO_STRING(_stState[_nStationId].State), ': ');
        f_MessageSet(_stMsg);
      END_IF
    END_IF

  //---------------------------------------------------------------------------
  // fatal errors
  //  - It's a Sin..
  //  - That went south so fast.
  //  - Wasn't expecting that..
  //---------------------------------------------------------------------------
  E_STATION_STATE.STATION_ERROR_LIST_GET_HEAD_FAULT,
  E_STATION_STATE.STATION_ERROR_LIST_REMOVE_HEAD_FAULT,
  E_STATION_STATE.STATION_ERROR_LIST_ADD_TAIL_FAULT,
  E_STATION_STATE.STATION_ERROR_LIST_MOVER_ID_INVALID:
    // yes, but why?
    // cannot be fixed by ctrl
    _eFatalError                      := _stState[_nStationId].State;

    // leave the gun, take the cannoli
    _stState[_nStationId].State      := E_STATION_STATE.STATION_ERROR_FATAL;

    _stMsg.eType                      := E_MessageType.eMessageError;
    _stMsg.eSubdevice                 := Stationstate;
    _stMsg.iErrorNumber               := _stState[_nStationId].nMoverId;
    _stMsg.sText                      := concat(TO_STRING(_stState[_nStationId].State), ': ');
    _stMsg.sText                      := concat(_stMsg.sText, TO_STRING(_eFatalError));
    f_MessageSet(_stMsg);


  //---------------------------------------------------------------------------
  //---------------------------------------------------------------------------
  E_STATION_STATE.STATION_ERROR_FATAL:
    // repent, rethink, retry
    // State is dead. State remains dead: and we killed him!
    // There's no way out of here
    _sState                           := concat(TO_STRING(_stState[_nStationId].State), ': ');
    _sState                           := concat(_sState, TO_STRING(_eFatalError));
END_CASE
//-----------------------------------------------------------------------------
//-----------------------------------------------------------------------------
IF (_stState[_nStationId].nMoverId > 0) AND
   (_stState[_nStationId].nMoverId < MAX_MOVER+1)
THEN
  _stState[_nStationId].rMoverModPos  := _Mover[_stState[_nStationId].nMoverId].NcToPlc.ModuloActPos;
ELSE
  _stState[_nStationId].rMoverModPos  := 0.0;
END_IF
//-----------------------------------------------------------------------------
//-----------------------------------------------------------------------------
_stState[_nStationId].nQueue          := TO_USINT(_ItfStation[_nStationId].Count);
//-----------------------------------------------------------------------------
//-----------------------------------------------------------------------------
END_METHOD

PROPERTY DcTimeInSync : T_DCTIME64
GET
DcTimeInSync := _nDcTimeInSync;
END_GET
END_PROPERTY

METHOD MoveIn // prepares gearing in to MasterAxis
// get data from interface and calculate ModuloSyncPosition of Mover
_stInfeedGearData.iGearDenumerator      := _stStationGearData[_nStationId].iGearDenumerator;
_stInfeedGearData.rDeltaToMasterPos     := _stStationGearData[_nStationId].rDeltaToMasterPos;
_stInfeedGearData.rGearNumerator        := _stStationGearData[_nStationId].rGearNumerator;
_stInfeedGearData.rMasterStartDistance  := _stStationGearData[_nStationId].rMasterStartDistance;

// the modulo sync position does not come from the GearData struct, 
// because this value belongs to the station in this context. 
// The GearData struct is also used in the Ctrl/state pair of a mover, 
// this is an XOR use of GearInPosCA mechanics.
// This fb focus is on the station data
_rModuloSyncPosSlave                    := _stParameter[_nStationId].rPosWait
                                        +  _stParameter[_nStationId].rPosStop[_nNest]  // sidenote, synchronizing requires distance to get up to speed --> rPosStop > 0 is most helpful
                                        +  _stMoverData.rOffset
                                        +  _rMoverOffset[_nStationId][_stMoverData.nMoverId][_nNest];

_stInfeedGearData.rModuloSyncPosSlave   := _rModuloSyncPosSlave;

_stInfeed.rVelo                         := _stParameter[_nStationId].rVelo;
_stInfeed.rAcc                          := _stParameter[_nStationId].rAccDec;
_stInfeed.rJerk                         := _stParameter[_nStationId].rJerk;
_stInfeed.rGap                          := _stParameter[_nStationId].rGap;
_stInfeed.rDistance                     := _stParameter[_nStationId].rReleaseDistance;
_stInfeed.rDelta                        := TargetWindow;

// connect MasterAxis
_ItfMover[_stState[_nStationId].nMoverId].Master REF= _MasterAxis;

// init method
_ItfMover[_stState[_nStationId].nMoverId].GearInPosCa(FALSE, _stInfeed, _stInfeedGearData);

// clear substate
_eStateProgress           := E_PROGRESS.PROGRESS_INIT;
END_METHOD

PROPERTY StationGearData : REFERENCE TO ARRAY[1..MAX_STATION] OF ST_GEAR_DATA
SET
_stStationGearData REF= StationGearData;
END_SET
END_PROPERTY

END_FUNCTION_BLOCK

(* stored: Version 1.1.0.1, ProductVersion 3.1.4026.13
   POU fb_StationGearInPos: Id {19435571-e5f3-4c9b-9865-7e07690fce00}, SpecialFunc None
   Method Check: Id {8cd4d804-d4b8-499a-9efe-347b921dc270}
   Method Cycle: Id {9f6f1fa8-d6b2-498d-ad39-28a02983aa22}
   Property DcTimeInSync: Id {090a6f85-54cb-4059-bf22-52c348a89dab}
   Get Get: Id {e573ecf9-d257-44be-a2ae-f52bfd8acace}
   Method MoveIn: Id {366c3f40-530a-4188-a32f-7987d2de498b}
   Property StationGearData: Id {ec3f37e8-48f2-465a-b107-772a17ebd533}
   Set Set: Id {584f131d-8b50-4c21-b1f0-46dd6e6a18bc} *)
